PROGRAM MAIN
VAR
END_VAR

END_PROGRAM

(* stored: Version 1.1.0.1
   POU MAIN: Id {539e9fb6-405b-49fd-a7c0-88f52dcc4263} *)
